FUNCTION_BLOCK FB_TelescopeControl2
VAR_INPUT
	fbMachine	: FB_TelescopeMachine;
	bInit		: BOOL;
	bPark		: BOOL;
	bSlew		: BOOL;
	bTrack		: BOOL;
	bStop		: BOOL;
END_VAR
VAR_OUTPUT
END_VAR
VAR
	
END_VAR

fbMachine(
	bInit	:= bInit,
	bPark	:= bPark,
	bSlew 	:= bSlew,
	bTrack 	:= bTrack,
	bStop 	:= bStop
);

bInit	:= FALSE;
bPark	:= FALSE;
bSlew 	:= FALSE;
bTrack 	:= FALSE;
bStop 	:= FALSE;

END_FUNCTION_BLOCK

(* stored: Version 1.1.0.1, ProductVersion 3.1.4024.15
   POU FB_TelescopeControl2: Id {eddbf876-a986-4fe1-ba5b-16d782882b92}, SpecialFunc None *)
